// SIMATIC S7-200 project (STEP 7-Micro/WIN), CPU 221 REL 01.10

SYMBOL_TABLE USUARIO1
Inicio           I0.0     // NA
Paro             I0.1     // NC
Rele             I0.2     // NA
Nivel_max        I0.3     // NA
Nivel_min        I0.4     // NA
Motor            Q0.0
Elv2             Q0.1
Led_marcha       Q0.2
Led_bomba        Q0.3
Led_falla        Q0.4
END_SYMBOL_TABLE

ORGANIZATION_BLOCK PRINCIPAL:OB1
TITLE=COMENTARIOS DEL PROGRAMA
BEGIN
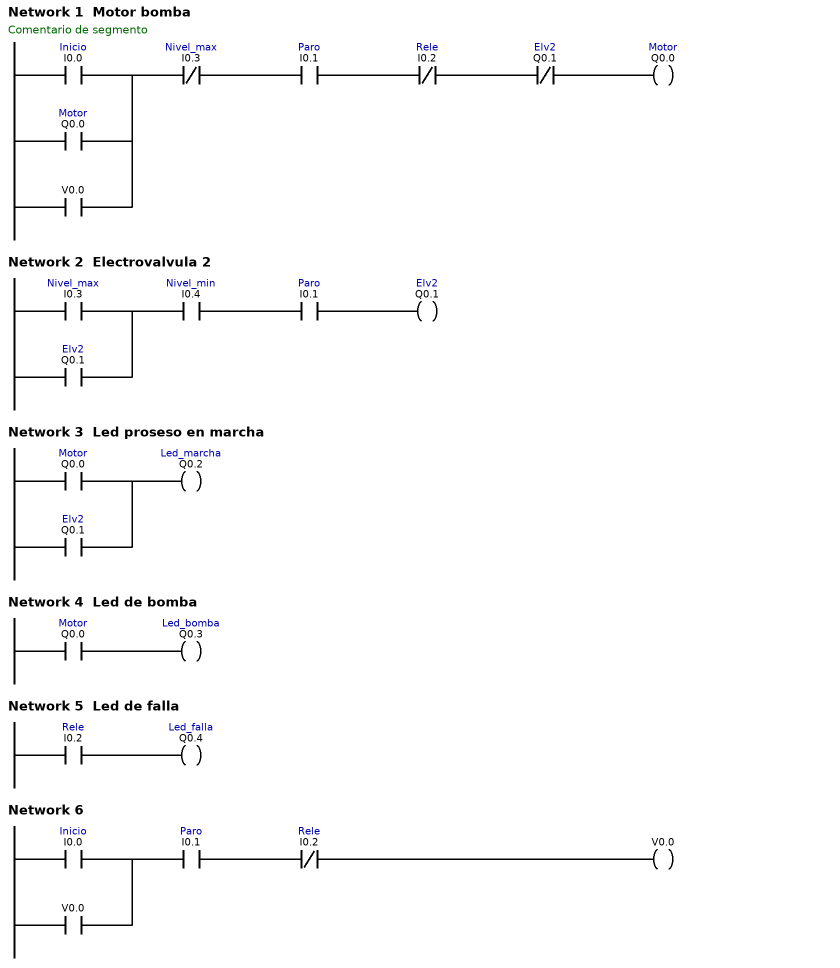
Network 1 // Motor bomba
// Comentario de segmento
// (network saved uncompiled; LAD cells follow)
// row 0: c0 -| |- Inicio:I0.0 v  c1 -|/|- Nivel_max:I0.3  c2 -| |- Paro:I0.1  c3 -|/|- Rele:I0.2  c4 -|/|- Elv2:Q0.1  c5 -( ) Motor:Q0.0
// row 1: c0 -| |- Motor:Q0.0 ^v
// row 2: c0 -| |- V0.0 ^
Network 2 // Electrovalvula 2
LD     Nivel_max:I0.3
O      Elv2:Q0.1
A      Nivel_min:I0.4
A      Paro:I0.1
=      Elv2:Q0.1
Network 3 // Led proseso en marcha
// (network saved uncompiled; LAD cells follow)
// row 0: c0 -| |- Motor:Q0.0 v  c1 -( ) Led_marcha:Q0.2
// row 1: c0 -| |- Elv2:Q0.1 ^
Network 4 // Led de bomba
LD     Motor:Q0.0
=      Led_bomba:Q0.3
Network 5 // Led de falla
LD     Rele:I0.2
=      Led_falla:Q0.4
Network 6
// (network saved uncompiled; LAD cells follow)
// row 0: c0 -| |- Inicio:I0.0 v  c1 -| |- Paro:I0.1  c2 -|/|- Rele:I0.2  c3 --  c4 --  c5 -( ) V0.0
// row 1: c0 -| |- V0.0 ^
END_ORGANIZATION_BLOCK
